PROGRAM P_FeedForward
VAR
	fbFF : FB_FeedForward;
END_VAR

IF (G_Enables.bEnableFF AND G_Mode.bRunning) THEN
fbFF(
	fXDotRef := G_OPC.fXDotRef,
	fQMaxUp := G_Parameter.fQMaxUp,
	fQMaxDown := G_Parameter.fQMaxDown,
	fDeadUp := G_Parameter.fDeadUp,
	fDeadDown := G_Parameter.fDeadDown,
	
	fPa := G_OPC.fPaLowerFiltered,
	fPb := G_OPC.fPbFiltered,
	fPs := G_OPC.fPsFiltered,
	
	fUFF => G_OPC.fUFF
);
END_IF

END_PROGRAM

(* stored: Version 1.1.0.1, ProductVersion 3.1.4024.12
   POU P_FeedForward: Id {202d862f-f86c-42e9-b9cf-42d47a621534}, SpecialFunc None *)
